# B&R Automation Studio project PlcProject
Automation Studio 4.9

## Configuration EM0611

CPU X20EM0611, AutomationRuntime 6.0.2, Build 11.3.0, Vc 6.0.0

### Task classes (Cpu.sw)
```
Cyclic#3 (cycle 4000 us, tolerance 0 us):
  Program <- Program.prg
  ProcCtrl <- ProcCtrl.prg
Binaries: udbdef, FWRules, TCData, sysconf, Role, User, iomap, ashwd, BRRole, asfw, arconfig, ashwac, UaCsConfig
Libraries: MTBasics, runtime, brsystem, sys_lib, MTTypes, MTProfile, astime, AsIecCon, Utils
```

### Hardware
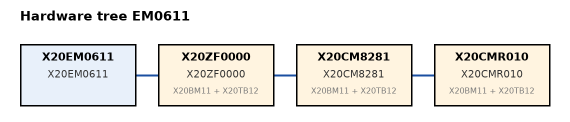
```
X20BM11 : X20BM11 v1.1.0.0  [X2X1 -> X20EM0611.IF6]
X20BM11_a : X20BM11 v1.1.0.0  [X2X1 -> X20BM11.X2X2]
X20BM11_b : X20BM11 v1.1.0.0  [X2X1 -> X20BM11_a.X2X2]
X20CM8281 : X20CM8281 v1.5.0.0  [SS1 -> X20TB12_a.SS; SL -> X20BM11_a.SL1]
  Supervision = off
X20CMR010 : X20CMR010 v1.4.2.0  [SS1 -> X20TB12_b.SS; SL -> X20BM11_b.SL1]
  Supervision = off
  DatapointInfoEnable = on
  OperatingDataEnable = on
  RelHumInfoEnable = on
  TempInfoEnable = on
X20EM0611 : X20EM0611 v1.1.1.0
  Connector IF2:
    ActivateDevice = 1
    HostName = cg-automation
    Mode = Manual
    InternetAddress = 192.168.1.50
    SubnetMask = 255.255.255.0
    ActivateSnmp = 1
  Connector IF3:
    EplHostName = cg-automation
    CycleTime = 800
    HostName = cg-automation
  ConfigurationID = OpcUaLogDemo_EM0611
  EnableUsbRemoteInstall = 1
  TimerDeviceType = EPLX2X
  TimerDevice = X20EM0611.IF3
  IdleTaskClass = 4
  TaskClassIdleTime = 2400
  Cyclic1Duration = 800
  Cyclic1Tolerance = 0
  Cyclic2Duration = 2400
  Cyclic2Tolerance = 0
  Cyclic3Duration = 4000
  Cyclic3Tolerance = 0
  Cyclic8Duration = 9600
  FileDevice1
  FileDeviceName1 = USER
  FileDevicePath1 = USER_PATH
  EthernetHostName = cg-automation
  ActivateFtpServer = 1
  FTPProtocol = 1
  FtpUser1
  FtpUsername1 = PLC
  FtpUserPassword1 = bDesm58/cQRkURzOhN7y21+dfhrAC+sJ92qeVEDnjI0=  // admin
  FtpUserSalt1 = O6GTINpH
  FTPAccessRight1 = 0
  ActivateWebServer = 1
  ActivateSdm = 1
X20TB12 : X20TB12 v1.0.0.0
X20TB12_a : X20TB12 v1.0.0.0
X20TB12_b : X20TB12 v1.0.0.0
X20ZF0000 : X20ZF0000 v1.2.2.0  [SS1 -> X20TB12.SS; SL -> X20BM11.SL1]
```

## Logical view

Binary libraries used (declarations not repeated): operator, runtime, AsIecCon, astime, MTBasics 6.0.0, brsystem, sys_lib, MTTypes, MTProfile 6.0.0

### Package Logical/Libraries - Global libraries

### Library Logical/Libraries/Utils (ANSIC)

#### Utils.fun - Exported functions and function blocks
```iecst
{REDUND_ERROR} FUNCTION f_Random : INT (*TODO: Add your comment here*) (*$GROUP=User,$CAT=User,$GROUPICON=User.png,$CATICON=User.png*)
END_FUNCTION
```

#### f_Random.c
```c
#include <bur/plctypes.h>
#ifdef __cplusplus
	extern "C"
	{
#endif
	#include "Utils.h"
#ifdef __cplusplus
	};
#endif
/* TODO: Add your comment here */
signed short f_Random(void)
{
	/*TODO: Add your code here*/
	return rand();
}
```

### Program Logical/ProcCtrl (IEC)

#### Types.typ
```iecst
TYPE
	tstProcessSim : 	STRUCT
		rDelayTime : REAL;
		rGain : REAL;
		rTimeConstant : REAL;
	END_STRUCT;
END_TYPE
```

#### Variables.var
```iecst
VAR
	fbPid : MTBasicsPID;
	rActValue : REAL;
	rSetValue : REAL;
	fbDelay : MTBasicsTimeDelay;
	fbPT1 : MTBasicsPT1;
	stProcessSimConfig : tstProcessSim;
	stPidPar : MTPIDParametersType;
	rCount : REAL;
	rValue : REAL;
	iRandom : ARRAY[0..4] OF INT;
END_VAR
(*Simulation*)
VAR
	dtUtcTime : DATE_AND_TIME;
	fbUtcDTGetTime : UtcDTGetTime;
	fbRtInfo : RTInfo;
	udiCycleTime_us : UDINT;
	udiTimeCount_us : UDINT;
END_VAR
VAR CONSTANT
	rPI : REAL := 3.14159;
END_VAR
VAR
	rTimeCount_s : REAL;
	rTest : REAL;
END_VAR
(*Simulation Values*)
VAR
	diState : DINT;
END_VAR
VAR CONSTANT
	diSTATE_STOPPED : DINT := 0;
	diSTATE_RUNNING : DINT := 10;
END_VAR
VAR
	fbMtBasicLimiter : MTBasicsLimiter;
	rActVelocity : REAL;
	rMotorTemp : REAL;
	iMaxStopTime : INT;
	iMaxRunTime : INT;
END_VAR
```

#### Cyclic.st
```iecst
PROGRAM _CYCLIC
	(* Insert code here *)
	udiTimeCount_us := udiTimeCount_us + udiCycleTime_us;
	rTimeCount_s := udiTimeCount_us / 1000000.0;

	rCount := rCount + 0.01;

//	rTest := SIN(rTimeCount_s * 2 * rPI * rPeriode_s);

	fbPid.ActValue := rActValue;
	fbPid.SetValue := rSetValue;// + SIN(rCount);
	fbPid.PIDParameters := stPidPar;
	fbPid.MinOut := -50;
	fbPid.MaxOut := 50;
	fbPid.Enable := TRUE;
	fbPid();

	fbDelay.In := fbPid.Out;
	fbDelay.InitialValue := 0;
	fbDelay.DelayTime := stProcessSimConfig.rDelayTime;
	fbDelay.Enable := TRUE;
	fbDelay();

	fbPT1.In := fbDelay.Out;
	fbPT1.Gain := stProcessSimConfig.rGain;
	fbPT1.TimeConstant := stProcessSimConfig.rTimeConstant;
	fbPT1.Enable := TRUE;
	fbPT1();

	rActValue := fbPT1.Out;

	iRandom[0] := f_Random();
	iRandom[1] := f_Random();
	iRandom[2] := f_Random();
	iRandom[3] := f_Random();
	iRandom[4] := f_Random();

	fbMtBasicLimiter.Enable := TRUE;

	CASE diState OF

		diSTATE_STOPPED:

			fbMtBasicLimiter.In := 0;

			rActVelocity := fbMtBasicLimiter.Out;

			IF (REAL_TO_DINT(rTimeCount_s) MOD iMaxStopTime) = 0 THEN
				diState := diSTATE_RUNNING;
				iMaxRunTime := (f_Random() MOD 101) + 120; // value between 120...221
			END_IF

		diSTATE_RUNNING:

			fbMtBasicLimiter.In := 1500;

			rActVelocity := fbMtBasicLimiter.Out
			+ (SIN(rTimeCount_s * 2 * rPI / 10) * 20) // Periode 20s, Amplitude 100
			+ f_Random() MOD 30; // Random-Wert +-30

			IF (REAL_TO_DINT(rTimeCount_s) MOD iMaxRunTime) = 0 THEN
				diState := diSTATE_STOPPED;
				iMaxStopTime := (f_Random() MOD 60) + 60; //value between 20...43
			END_IF

		ELSE
			;
	END_CASE

	IF rActVelocity <> 0 THEN
		rMotorTemp := rMotorTemp + (75 - rMotorTemp) * 0.0001; // heating
	ELSE
		rMotorTemp := rMotorTemp - (rMotorTemp - 20) * 0.00005; // cool down
	END_IF

	fbMtBasicLimiter();
END_PROGRAM
```

#### Init.st
```iecst
PROGRAM _INIT
	(* Insert code here *)
	stProcessSimConfig.rDelayTime := 0.5;
	stProcessSimConfig.rGain := 0.9;
	stProcessSimConfig.rTimeConstant := 5;

	iMaxStopTime := 5; //5s init value

	stPidPar.DerivativeTime := 0;
	stPidPar.FilterTime := 0;
	stPidPar.Gain := 2;
	stPidPar.IntegrationTime := 10;

	fbRtInfo(enable := TRUE);
	udiCycleTime_us := fbRtInfo.cycle_time;

	fbMtBasicLimiter.MaxNegSlewRate := 250;
	fbMtBasicLimiter.MaxPosSlewRate := 350;
	fbMtBasicLimiter.MinOut := 0;
	fbMtBasicLimiter.MaxOut := 1500;

END_PROGRAM
```

### Program Logical/Program (IEC)

#### Variables.var
```iecst
VAR
	rCount : {REDUND_UNREPLICABLE} REAL := 0.0;
	rSine : REAL;
END_VAR
```

#### Cyclic.st
```iecst
PROGRAM _CYCLIC
	(* Insert code here *)
	rCount := rCount + 0.1;
	rSine := SIN(rCount);
END_PROGRAM
```

Listed in the project but not available here: Logical/Global.typ, Logical/Global.var, Logical/Libraries/Utils/Types.typ, Logical/Libraries/Utils/Constants.var
